INTERFACE I_PtInterval

METHOD inMonth : DINT
VAR_INPUT
END_VAR
END_METHOD

METHOD inYears : DINT
VAR_INPUT
END_VAR
END_METHOD

END_INTERFACE

(* stored: Version 1.1.0.1, ProductVersion 3.1.4024.12
   Itf I_PtInterval: Id {7eb7558e-4186-43f6-827a-bf1a6c972e8f}
   Method inMonth: Id {82085986-cc9e-4b47-9546-54f8ea9d238f}
   Method inYears: Id {c6e79af5-8c14-4568-9b6f-c8872f07cf34} *)
